// Mitsubishi GX Works2 project: PLC IO Test   PLC: Q03UD
// PLC Unity Connect Test

PROGRAM MAIN
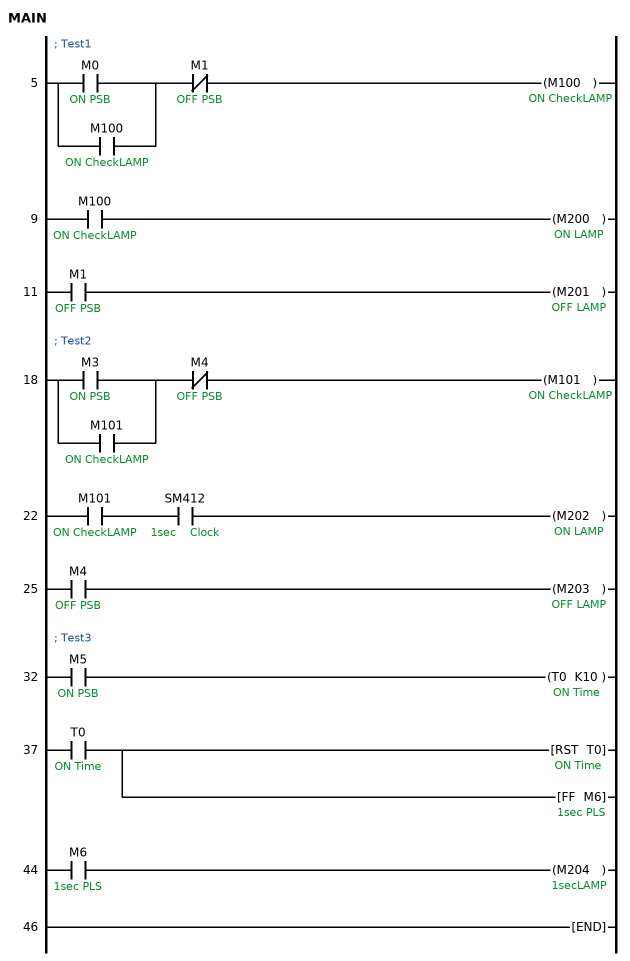
; Test1
5     LD      M0  ; ON PSB
      OR      M100  ; ON CheckLAMP
      ANI     M1  ; OFF PSB
      OUT     M100  ; ON CheckLAMP
9     LD      M100  ; ON CheckLAMP
      OUT     M200  ; ON LAMP
11    LD      M1  ; OFF PSB
      OUT     M201  ; OFF LAMP
; Test2
18    LD      M3  ; ON PSB
      OR      M101  ; ON CheckLAMP
      ANI     M4  ; OFF PSB
      OUT     M101  ; ON CheckLAMP
22    LD      M101  ; ON CheckLAMP
      AND     SM412  ; 1sec    Clock
      OUT     M202  ; ON LAMP
25    LD      M4  ; OFF PSB
      OUT     M203  ; OFF LAMP
; Test3
32    LD      M5  ; ON PSB
      OUT     T0 K10  ; ON Time
37    LD      T0  ; ON Time
      RST     T0  ; ON Time
      FF      M6  ; 1sec PLS
44    LD      M6  ; 1sec PLS
      OUT     M204  ; 1secLAMP
46    END
END_PROGRAM

// device comments not shown above
M102  ; ON Check
T1  ; OFF Time
